{attribute 'qualified_CLOSEly'}
VAR_GLOBAL
	
I_INDEXING_22_GRIPPER_CLOSE_1 AT %I* : BOOL;
I_INDEXING_2_GRIPPER_CLOSE_2 AT %I* : BOOL;
I_INDEXING_2_GRIPPER_CLOSE_3 AT %I* : BOOL;
I_INDEXING_2_GRIPPER_CLOSE_4 AT %I* : BOOL;
I_INDEXING_2_GRIPPER_OPEN_1 AT %I* : BOOL;
I_INDEXING_2_GRIPPER_OPEN_2 AT %I* : BOOL;
I_INDEXING_2_GRIPPER_OPEN_3 AT %I* : BOOL;
I_INDEXING_2_GRIPPER_OPEN_4 AT %I* : BOOL;
I_INDEXING_2_GRIPPER_EXT_UP AT %I* : BOOL;
I_INDEXING_2_GRIPPER_EXT_DOWN AT %I* : BOOL;

O_INDEXING_2_GRIPPER_EXT_UP AT %Q* : BOOL;
O_INDEXING_2_GRIPPER_EXT_DOWN AT %Q* : BOOL;
O_INDEXING_2_GRIPPER_CLOSE_1 AT %Q* : BOOL;
O_INDEXING_2_GRIPPER_CLOSE_2 AT %Q* : BOOL;
O_INDEXING_2_GRIPPER_CLOSE_3 AT %Q* : BOOL;
O_INDEXING_2_GRIPPER_CLOSE_4 AT %Q* : BOOL;
O_INDEXING_2_GRIPPER_OPEN_1 AT %Q* : BOOL;
O_INDEXING_2_GRIPPER_OPEN_2 AT %Q* : BOOL;
O_INDEXING_2_GRIPPER_OPEN_3 AT %Q* : BOOL;
O_INDEXING_2_GRIPPER_OPEN_4 AT %Q* : BOOL;

I_PRESS_STOPPER_DOWN AT %I* : BOOL;
I_PRESS_STOPPER_UP AT %I* : BOOL;

O_PRESS_STOPPER_DOWN AT %Q* : BOOL;
O_PRESS_STOPPER_UP AT %Q* : BOOL;

O_INDEXING_HOME   : BOOL;
O_ROTATION_DONE : BOOL;
O_ROTATION_START : BOOL;
O_ROTATION_STOP : BOOL;

I_INDEXING_2_READY_FOR_STRAIGHTEN: BOOL;
I_INDEXING_2_HOME : BOOL;
O_INDEXING_2_POWER_OFF AT %Q* : BOOL;

I_INDEXING_2_ROTATION_DONE: BOOL :=TRUE;
I_ALL_GRIPPER_OPEN: BOOL;
NUMBER_OF_STRAIGHTEN: INT :=0;
INDEXING_2_CASE: INT ;
TOTALNUMBER_OF_STRAIGHTEN :INT :=1;
CARRIER_INDEX: BYTE;

DataByteOutput2 AT%Q* : ARRAY[0..7] OF BYTE;
DataByteInput2 AT%I* : ARRAY[0..7] OF BYTE;
END_VAR

(* stored: Version 1.1.0.1, ProductVersion 3.1.4020.12
   GVL INDEXING_2_VAR: Id {b58aeea9-68aa-41b4-8609-6c0fd87eeca8} *)
